// TIA Portal V20 export
// export: Created 2026-04-11T06:02:30.1926236Z, ExportSetting WithDefaults, DisplayName Totally Integrated Automation Portal, DisplayVersion V20, DisplayName TIA Portal Openness, DisplayVersion V20, DisplayName TIA Portal Version Control Interface, DisplayVersion V20, DisplayName STEP 7 Professional, DisplayVersion V20, DisplayName STEP 7 Safety, DisplayVersion V20, DisplayName WinCC Basic/Comfort/Advanced, DisplayVersion V20, DisplayName WinCC Unified, DisplayVersion V20
TYPE "udtHMI_DigitalInput"
// stored: IsFailsafeCompliant false
   STRUCT
      iMode : Int;   // Current mode
      bOn { ExternalWritable := 'False'} : Bool;   // Status of the sensor
      bOnActual { ExternalWritable := 'False'} : Bool;   // Status of the physical sensor
      bPB_On : Bool;   // Turn input on in manual mode
      bPB_Off : Bool;   // Turn input off in manual mode
      bPBEN_On { ExternalWritable := 'False'} : Bool;   // Enable manual mode on push button
      bPBEN_Off { ExternalWritable := 'False'} : Bool;   // Enable manual mode off push button
   END_STRUCT;
END_TYPE
